FUNCTION_BLOCK Estocagem_Lodo (* Composite Function Block Type *)
  (* Standard: 61499-2 *)
  (* Version 0.0, 28/04/2026, template *)
  PACKAGE Hidryco.HidrycoLib;
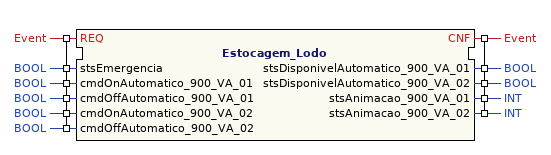
  EVENT_INPUT
    REQ WITH cmdOnAutomatico_900_VA_01, cmdOffAutomatico_900_VA_01, cmdOnAutomatico_900_VA_02, cmdOffAutomatico_900_VA_02, stsEmergencia; (* Normal Execution Request *)
  END_EVENT
  EVENT_OUTPUT
    CNF WITH stsDisponivelAutomatico_900_VA_01, stsDisponivelAutomatico_900_VA_02, stsAnimacao_900_VA_02, stsAnimacao_900_VA_01; (* Execution Confirmation *)
  END_EVENT
  VAR_INPUT
    stsEmergencia : BOOL;
    cmdOnAutomatico_900_VA_01 : BOOL;
    cmdOffAutomatico_900_VA_01 : BOOL;
    cmdOnAutomatico_900_VA_02 : BOOL;
    cmdOffAutomatico_900_VA_02 : BOOL;
  END_VAR
  VAR_OUTPUT
    stsDisponivelAutomatico_900_VA_01 : BOOL;
    stsDisponivelAutomatico_900_VA_02 : BOOL;
    stsAnimacao_900_VA_01 : INT;
    stsAnimacao_900_VA_02 : INT;
  END_VAR
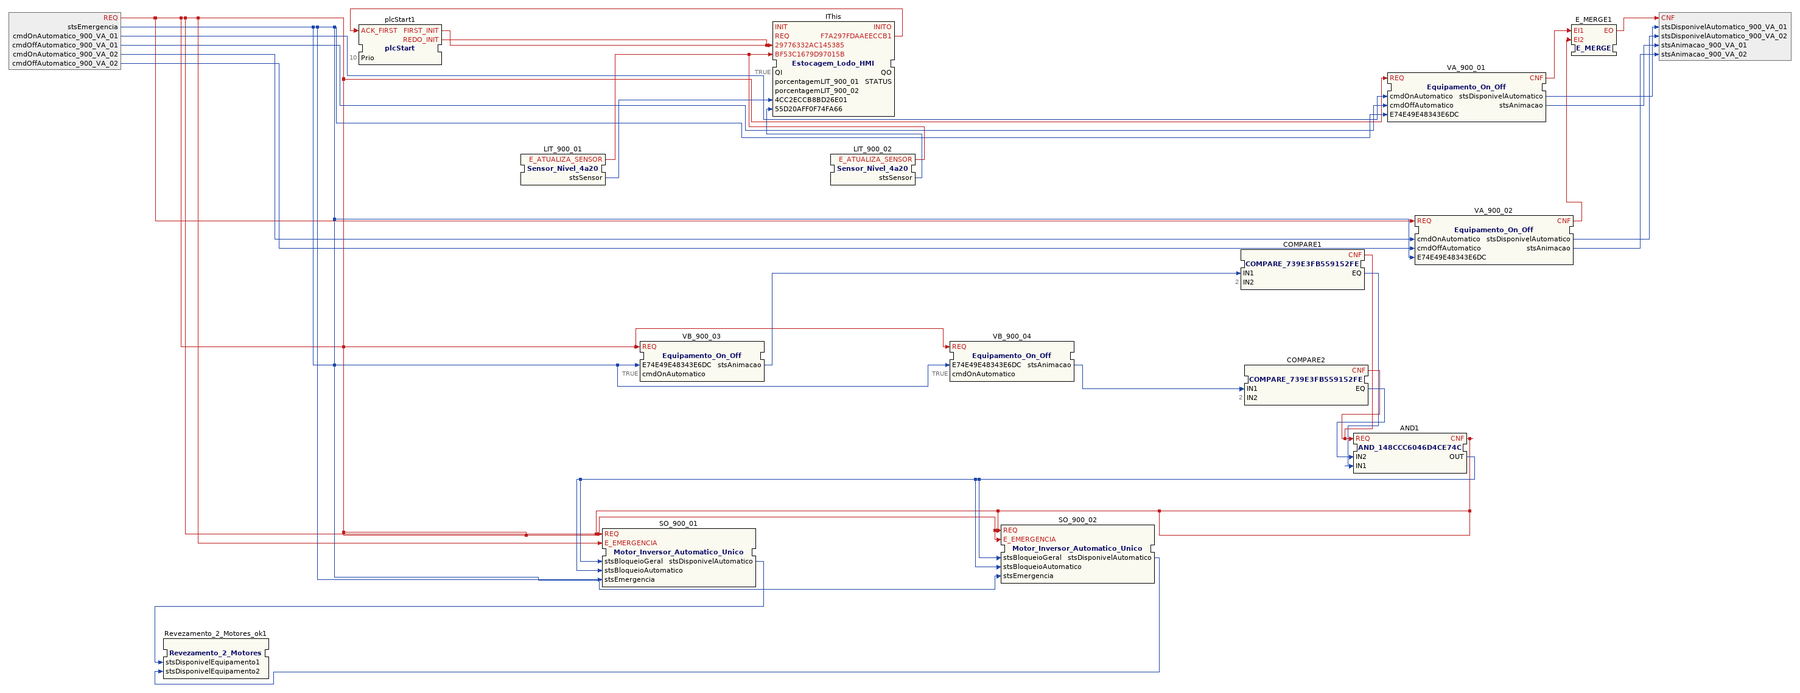
  FBS
    LIT_900_02 : Sensor_Nivel_4a20;
    LIT_900_01 : Sensor_Nivel_4a20;
    VA_900_01 : Equipamento_On_Off;
    VA_900_02 : Equipamento_On_Off;
    VB_900_03 : Equipamento_On_Off(cmdOnAutomatico := TRUE);
    VB_900_04 : Equipamento_On_Off(cmdOnAutomatico := TRUE);
    SO_900_01 : Motor_Inversor_Automatico_Unico;
    SO_900_02 : Motor_Inversor_Automatico_Unico;
    Revezamento_2_Motores_ok1 : Revezamento_2_Motores;
    COMPARE1 : COMPARE_739E3FB559152FE(IN2 := 2); {SET_ATTRIBUTE(Configuration.GenericFBType.InterfaceParams, Runtime.Standard#CNT:=2;IN${CNT$}:INT)}
    COMPARE2 : COMPARE_739E3FB559152FE(IN2 := 2); {SET_ATTRIBUTE(Configuration.GenericFBType.InterfaceParams, Runtime.Standard#CNT:=2;IN${CNT$}:INT)}
    AND1 : AND_148CCC6046D4CE74C; {SET_ATTRIBUTE(Configuration.GenericFBType.InterfaceParams, Runtime.Standard#CNT:=2)}
    IThis : Estocagem_Lodo_HMI(QI := TRUE);
    plcStart1 : plcStart(Prio := 10);
    E_MERGE1 : E_MERGE;
  END_FBS
  EVENT_CONNECTIONS
    COMPARE2.CNF TO AND1.REQ;
    COMPARE1.CNF TO AND1.REQ;
    VA_900_01.CNF TO E_MERGE1.EI1;
    VA_900_02.CNF TO E_MERGE1.EI2;
    E_MERGE1.EO TO CNF;
    REQ TO VA_900_01.REQ;
    REQ TO VA_900_02.REQ;
    plcStart1.FIRST_INIT TO IThis.29776332AC145385;
    plcStart1.REDO_INIT TO IThis.29776332AC145385;
    LIT_900_01.E_ATUALIZA_SENSOR TO IThis.BF53C1679D97015B;
    LIT_900_02.E_ATUALIZA_SENSOR TO IThis.BF53C1679D97015B;
    IThis.F7A297FDAAEECCB1 TO plcStart1.ACK_FIRST;
    REQ TO VB_900_03.REQ;
    REQ TO SO_900_01.REQ;
    REQ TO VB_900_04.REQ;
    REQ TO SO_900_02.REQ;
    REQ TO SO_900_01.E_EMERGENCIA;
    REQ TO SO_900_02.E_EMERGENCIA;
    AND1.CNF TO SO_900_02.REQ;
    AND1.CNF TO SO_900_01.REQ;
  END_CONNECTIONS
  DATA_CONNECTIONS
    SO_900_01.stsDisponivelAutomatico TO Revezamento_2_Motores_ok1.stsDisponivelEquipamento1;
    SO_900_02.stsDisponivelAutomatico TO Revezamento_2_Motores_ok1.stsDisponivelEquipamento2;
    VB_900_04.stsAnimacao TO COMPARE2.IN1;
    COMPARE2.EQ TO AND1.IN2;
    VB_900_03.stsAnimacao TO COMPARE1.IN1;
    COMPARE1.EQ TO AND1.IN1;
    AND1.OUT TO SO_900_02.stsBloqueioGeral;
    AND1.OUT TO SO_900_02.stsBloqueioAutomatico;
    AND1.OUT TO SO_900_01.stsBloqueioGeral;
    AND1.OUT TO SO_900_01.stsBloqueioAutomatico;
    cmdOnAutomatico_900_VA_01 TO VA_900_01.cmdOnAutomatico;
    cmdOffAutomatico_900_VA_01 TO VA_900_01.cmdOffAutomatico;
    VA_900_01.stsDisponivelAutomatico TO stsDisponivelAutomatico_900_VA_01;
    VA_900_02.stsDisponivelAutomatico TO stsDisponivelAutomatico_900_VA_02;
    cmdOnAutomatico_900_VA_02 TO VA_900_02.cmdOnAutomatico;
    cmdOffAutomatico_900_VA_02 TO VA_900_02.cmdOffAutomatico;
    VA_900_02.stsAnimacao TO stsAnimacao_900_VA_02;
    VA_900_01.stsAnimacao TO stsAnimacao_900_VA_01;
    LIT_900_01.stsSensor TO IThis.4CC2ECCB8BD26E01;
    LIT_900_02.stsSensor TO IThis.55D20AFF0F74FA66;
    stsEmergencia TO VA_900_01.E74E49E48343E6DC;
    stsEmergencia TO VA_900_02.E74E49E48343E6DC;
    stsEmergencia TO VB_900_04.E74E49E48343E6DC;
    stsEmergencia TO VB_900_03.E74E49E48343E6DC;
    stsEmergencia TO SO_900_01.stsEmergencia;
    stsEmergencia TO SO_900_02.stsEmergencia;
  END_CONNECTIONS
END_FUNCTION_BLOCK
